// Upper bounds of devices
VAR_GLOBAL CONSTANT
    cUpperBoundSafetyTestTrolley    : UINT := 4;
END_VAR

VAR_GLOBAL
    {attribute 'TcContextName':='MainTask'}
    SafetyTestTrolley   : ARRAY [0..cUpperBoundSafetyTestTrolley] OF FB_SafetyTestTrolley;
END_VAR

(* stored: Version 1.1.0.1, ProductVersion 3.1.4024.12
   GVL MachineObjectsArray: Id {4c315092-3eb0-4ba7-8ac2-d1189a2ec0e3} *)
